// TIA Portal V16 export
// export: Created 2023-04-18T08:26:50.8983284Z, ExportSetting WithDefaults, DisplayName Totally Integrated Automation Portal, DisplayVersion V16, DisplayName TIA Portal Version Control Interface, DisplayVersion V16, DisplayName TIA Portal Openness, DisplayVersion V16, DisplayName SINAMICS Startdrive Advanced, DisplayVersion V16, DisplayName SINAMICS Startdrive G130, G150, S120, S150, SINAMICS MV, S210, DisplayVersion V16, DisplayName SINAMICS Startdrive G110M, G120, G120C, G120D, G120P, DisplayVersion V16, DisplayName STEP 7 Professional, DisplayVersion V16, DisplayName SIMATIC Energy Suite, DisplayVersion V16, DisplayName STEP 7 Safety, DisplayVersion V16, DisplayName WinCC Professional, DisplayVersion V16, DisplayName SIMATIC Visualization Architect, DisplayVersion V16
FUNCTION_BLOCK "IEQ"   // FB9, LAD
{ S7_Optimized_Access := 'TRUE' }
VERSION : 0.1
// stored: AutoNumber true, IsIECCheckEnabled false, IsRetainMemResEnabled false, MemoryReserve 100, SetENOAutomatically false, UDAEnableTagReadback false
   VAR_INPUT
      Fusible_R : Bool;
      Fusible_S : Bool;
      Fusible_T : Bool;
      "Fallo_ Tarjeta" : Bool;
      Seta : Bool;
      Fallo_Red : Bool;
      Ahorro_S0 : Bool;
      Ahorro_S1 : Bool;
      Directo_S0 : Bool;
      Directo_S1 : Bool;
      Nucleo_S0 : Bool;
      Nucleo_S1 : Bool;
      Tiristor : Int;
      Nucleo : Int;
   END_VAR
   VAR_OUTPUT
      alpha : Int;
      ventiladores : Bool;
      Ahorro_P0 : Bool;
      Ahorro_P1 : Bool;
      Directo_P0 : Bool;
      Directo_P1 : Bool;
      Nucleo_P0 : Bool;
      Nucleo_P1 : Bool;
   END_VAR
   VAR_IN_OUT
      AHM1 : "AHM1";
      IEQ : "IEQSY";
   END_VAR
   VAR
      Etapa_Emergencia : Int;
      Alpha_Conmutación : Bool;
   END_VAR
   VAR RETAIN
      Etapa : Int;
   END_VAR
   VAR
      S_Etapa : Int;
      Error : Int;
      Temporizadores : Struct
         T_E1 { S7_SetPoint := 'True'} : TON_TIME;
         T_E2 { S7_SetPoint := 'True'} : TON_TIME;
         T_E3 { S7_SetPoint := 'True'} : TON_TIME;
         T_E4 { S7_SetPoint := 'True'} : TON_TIME;
         T_E5 { S7_SetPoint := 'True'} : TON_TIME;
         T_E7 { S7_SetPoint := 'True'} : TON_TIME;
         T_SE1 { S7_SetPoint := 'True'} : TON_TIME;
         T_SE2 { S7_SetPoint := 'True'} : TON_TIME;
         T_SE3 { S7_SetPoint := 'True'} : TON_TIME;
         T_SE4 { S7_SetPoint := 'True'} : TON_TIME;
      END_STRUCT;
      F_TRIG_Seta { S7_SetPoint := 'True'} : F_TRIG;
      F_TRIG_Fusible_R { S7_SetPoint := 'True'} : F_TRIG;
      F_TRIG_Fusible_S { S7_SetPoint := 'True'} : F_TRIG;
      F_TRIG_Fusible_T { S7_SetPoint := 'True'} : F_TRIG;
      F_TRIG_Fallo_Red { S7_SetPoint := 'True'} : F_TRIG;
      R_TRIG_ETAPA { S7_SetPoint := 'True'} : R_TRIG;
      R_TRIG_BTN { S7_SetPoint := 'True'} : R_TRIG;
      F_TRIG_BTN { S7_SetPoint := 'True'} : F_TRIG;
      NormVal { ExternalAccessible := 'False'; ExternalVisible := 'False'; ExternalWritable := 'False'} : Real;
      message : String;
      showPopUp : Bool;
      ValHMI { ExternalAccessible := 'False'; ExternalVisible := 'False'; ExternalWritable := 'False'} : Int;
   END_VAR
BEGIN

REGION Network 1 (SCL)
   //*********************************************************************************************************************
   // Autor : Illya Kulinich
   // 
   // Descripción : 

   //*********************************************************************************************************************
END_REGION

REGION Network 2 (SCL): Flancos

   #F_TRIG_Seta(CLK :=#Seta);
   #F_TRIG_Fusible_R(CLK := #Fusible_R);
   #F_TRIG_Fusible_S(CLK := #Fusible_S);
   #F_TRIG_Fusible_T(CLK := #Fusible_T);
   #F_TRIG_Fallo_Red(CLK := #Fallo_Red);
   #R_TRIG_BTN(CLK:=#IEQ.Conmutación.BTN);
   #F_TRIG_BTN(CLK := #IEQ.Conmutación.BTN);
END_REGION

REGION Network 3 (SCL): Conversión de temperatura en real

   #IEQ.Temperatura.Tiristores := (INT_TO_REAL(#Tiristor)) * 0.1;
   #IEQ.Temperatura.Nucleo  := (INT_TO_REAL(#Nucleo)) * 0.1;
END_REGION

REGION Network 4 (SCL): Declaración de temporizadores

       //
       #Temporizadores.T_SE1(IN := #Etapa_Emergencia = 1,
                             PT := T#1S);
       #Temporizadores.T_SE2(IN := #Etapa_Emergencia = 2,
                             PT := T#1S);
       #Temporizadores.T_SE3(IN := #Etapa_Emergencia = 3,
                             PT := T#1S);
       #Temporizadores.T_SE4(IN := #Etapa_Emergencia = 4,
                             PT := T#1S);

       //******************************************************************     
       #Temporizadores.T_E1(IN := #Etapa = 1,
                             PT := T#2.5s);
       #Temporizadores.T_E2(IN := #Etapa = 2,
                             PT := T#2.5s);
       #Temporizadores.T_E3(IN := #Etapa = 3,
                             PT := T#2.5s);
       #Temporizadores.T_E4(IN := #Etapa = 4,
                             PT := T#2.5s);
       #Temporizadores.T_E5(IN := #Etapa = 5,
                             PT := T#2.5s);
       #Temporizadores.T_E7(IN := #Etapa = 7,
                             PT := T#2.5s);
END_REGION

REGION Network 5 (SCL): Estado de Conmutación
   // Ahorro
   IF #Ahorro_S0 = 0 AND #Ahorro_S1 = 1 AND
       #Directo_S0 = 1 AND #Directo_S1 = 0 AND
       #Nucleo_S0 = 0 AND #Nucleo_S1 = 1 THEN
       #IEQ.Conmutación.Status := 'Ahorro';
   END_IF;


   // transición
   IF #Ahorro_S0 = 0 AND #Ahorro_S1 = 1 AND
       #Directo_S0 = 0 AND #Directo_S1 = 1 AND
       #Nucleo_S0 = 0 AND #Nucleo_S1 = 1 THEN
       #IEQ.Conmutación.Status  := 'Conmutando...';
   END_IF;

   // Directo 
   IF #Ahorro_S0 = 1 AND #Ahorro_S1 = 0 AND
       #Directo_S0 = 0 AND #Directo_S1 = 1 AND
       #Nucleo_S0 = 1 AND #Nucleo_S1 = 0 THEN
       #IEQ.Conmutación.Status  := 'Directo';

   END_IF;
END_REGION

REGION Network 6 (SCL): Seguridad

   IF (#F_TRIG_Fusible_R.Q OR #F_TRIG_Fusible_S.Q OR #F_TRIG_Fusible_T.Q) AND  #IEQ.Conmutación.BTN = 1  THEN
       #Etapa_Emergencia := 99;

   END_IF;

   IF #F_TRIG_Seta.Q AND #IEQ.Conmutación.BTN= 1 THEN
       #Etapa_Emergencia := 99;
   END_IF;

   IF  #IEQ.Temperatura.Tiristores >= 75.0 OR  #IEQ.Temperatura.Nucleo >= 120.0 AND #IEQ.Conmutación.BTN = 1 THEN
       #Etapa_Emergencia := 99;

   END_IF;

   IF #F_TRIG_Fallo_Red.Q AND #IEQ.Conmutación.BTN= 1 THEN
       #Etapa_Emergencia := 99;
   END_IF;



   // IF NOT #Fusible_R OR NOT #Fusible_S OR NOT #Fusible_T OR
   //     NOT #Seta OR
   //     NOT #Fallo_Red OR
   //     NOT (#IEQ.Temperatura.Tiristores < 50.0 AND #IEQ.Temperatura.Nucleo < 60.0) THEN
   IF #Fallo_Red THEN
       #Error := 1;
       #message := 'Error en la red';
       // pop up fallo fusibles
       // DTL timestamp
   ELSE
       #Error := 0;
   END_IF;

   IF #Error = 1 THEN
       #IEQ.Conmutación.BTN := 0;
       #IEQ.Alpha.Input_Value := 100;
       #showPopUp := 1;
   ELSE
       #Error := 0;
   END_IF;


   (* IF NOT  #Fallo_Red  THEN
       #IEQ.Conmutación.BTN := 0;
       // pop up fallo de red 
       // DTL timestamp
   END_IF;

   (* IF #"Fallo_ Tarjeta" THEN
       #IEQ.Conmutación.BTN := 0;
       // pop up tarjeta de tiristores
       // DTL timestamp
   END_IF; *)

   IF NOT (  < 50.0  OR  #IEQ.Temperatura.Tiristores < 50.0  OR  < 50.0  AND #IEQ.Temperatura.Nucleo < 60.0) AND #IEQ.Conmutación.BTN =1 THEN
       #IEQ.Conmutación.BTN := 0;
       // pop up temperatura 
       // DTL timestamp
   END_IF;
   *)
END_REGION

REGION Network 7 (SCL): Secuencia de emergencia





       IF #Etapa_Emergencia = 99 THEN

           #Etapa := 0;
           #Etapa_Emergencia := 1;

           #IEQ.Conmutación.BTN := 0;
           #Alpha_Conmutación := 1;

           #Ahorro_P0 := 0;
           #Ahorro_P1 := 1;
           #Directo_P0 := 0;
           #Directo_P1 := 1;
           #Nucleo_P0 := 0;
           #Nucleo_P1 := 1;
       END_IF;

       IF #Etapa_Emergencia = 1 AND #Temporizadores.T_SE1.Q THEN
           #Etapa_Emergencia := 2;
           #Alpha_Conmutación := 1;
           #Ahorro_P0 := 1;
           #Ahorro_P1 := 0;
           #Directo_P0 := 0;
           #Directo_P1 := 1;
           #Nucleo_P0 := 0;
           #Nucleo_P1 := 1;
       END_IF;

       IF #Etapa_Emergencia = 2 AND #Temporizadores.T_SE2.Q THEN
           #Etapa_Emergencia := 3;
           #Alpha_Conmutación := 1;
           #Ahorro_P0 := 1;
           #Ahorro_P1 := 0;
           #Directo_P0 := 0;
           #Directo_P1 := 1;
           #Nucleo_P0 := 1;
           #Nucleo_P1 := 0;

       END_IF;

       IF #Etapa_Emergencia = 3 AND #Temporizadores.T_SE3.Q THEN
           #Etapa_Emergencia := 0;
           #Etapa := 3;
       END_IF;
END_REGION

REGION Network 8 (SCL): Conmutación


       IF #Etapa = 99 THEN
           #Etapa := 1;

           #Alpha_Conmutación := 1;
           #Ahorro_P0 := 0;
           #Ahorro_P1 := 1;
           #Directo_P0 := 0;
           #Directo_P1 := 1;
           #Nucleo_P0 := 0;
           #Nucleo_P1 := 1;

       END_IF;

       IF #Etapa = 1 AND #Temporizadores.T_E1.Q THEN
           #Etapa := 2;
           #Alpha_Conmutación := 1;
           #Ahorro_P0 := 1;
           #Ahorro_P1 := 0;
           #Directo_P0 := 0;
           #Directo_P1 := 1;
           #Nucleo_P0 := 0;
           #Nucleo_P1 := 1;
       END_IF;

       IF #Etapa = 2 AND #Temporizadores.T_E2.Q THEN // Directo
           #Etapa := 3;
           #Alpha_Conmutación := 1;
           #Ahorro_P0 := 1;
           #Ahorro_P1 := 0;
           #Directo_P0 := 0;
           #Directo_P1 := 1;
           #Nucleo_P0 := 1;
           #Nucleo_P1 := 0;


       END_IF;


       IF #Etapa = 3 AND #Temporizadores.T_E3.Q AND #R_TRIG_BTN.Q AND #Error = 0 THEN
           #Etapa := 4;
           #Alpha_Conmutación := 1;
           #Ahorro_P0 := 1;
           #Ahorro_P1 := 0;
           #Directo_P0 := 0;
           #Directo_P1 := 1;
           #Nucleo_P0 := 0;
           #Nucleo_P1 := 1;

       END_IF;

       IF #Etapa = 4 AND #Temporizadores.T_E4.Q THEN
           #Etapa := 5;
           #Alpha_Conmutación := 1;
           #Directo_P0 := 0;
           #Directo_P1 := 1;

           #Ahorro_P0 := 0;
           #Ahorro_P1 := 1;

           #Nucleo_P0 := 0;
           #Nucleo_P1 := 1;

       END_IF;

       IF #Etapa = 5 AND #Temporizadores.T_E5.Q THEN
           #Etapa := 6;
           #Alpha_Conmutación := 0;
           #Ahorro_P0 := 0;
           #Ahorro_P1 := 1;
           #Directo_P0 := 1;
           #Directo_P1 := 0;
           #Nucleo_P0 := 0;
           #Nucleo_P1 := 1;

       END_IF;

       IF #Etapa = 6 AND #F_TRIG_BTN.Q THEN
           #Etapa := 99;
           #Alpha_Conmutación := 1;
       END_IF;
END_REGION

REGION Network 9 (SCL)

   REGION Definición de las condiciones de protección frente a valores no desados

       // si alguna de estas condiciónes son verdaderas el alpha setpoint pasa a 100
       IF #Alpha_Conmutación = 0 AND
           (#AHM1."Parametros Basicos"."40007 - Tension y Energia".PF1 < #IEQ.Alpha.RestriccionesAlpha.PF_Min_Alpha OR
           #AHM1."Parametros Basicos"."40007 - Tension y Energia".PF2 < #IEQ.Alpha.RestriccionesAlpha.PF_Min_Alpha OR
           #AHM1."Parametros Basicos"."40007 - Tension y Energia".PF3 < #IEQ.Alpha.RestriccionesAlpha.PF_Min_Alpha OR

           #AHM1."Harmonic data"."40529 - Distorsion Armonica V y A"."THD-V1" > #IEQ.Alpha.RestriccionesAlpha.Thd_V_Max OR
           #AHM1."Harmonic data"."40529 - Distorsion Armonica V y A"."THD-V2" > #IEQ.Alpha.RestriccionesAlpha.Thd_V_Max OR
           #AHM1."Harmonic data"."40529 - Distorsion Armonica V y A"."THD-V3" > #IEQ.Alpha.RestriccionesAlpha.Thd_V_Max OR

           #AHM1."Harmonic data"."40529 - Distorsion Armonica V y A"."THD-I1" > #IEQ.Alpha.RestriccionesAlpha.Thd_A_Max OR
           #AHM1."Harmonic data"."40529 - Distorsion Armonica V y A"."THD-I2" > #IEQ.Alpha.RestriccionesAlpha.Thd_A_Max OR
           #AHM1."Harmonic data"."40529 - Distorsion Armonica V y A"."THD-I3" > #IEQ.Alpha.RestriccionesAlpha.Thd_A_Max)
       THEN
           ;
           // si el pf y el thd en voltaje y corriente baja de x   alpha entra en error pon el valor a 100 ->  alpha a 100% = 5 V = 13834

           #IEQ.Alpha.AlphaEntero := 27648;
           #IEQ.Alpha.Status := 'Condiciones de red no se cumplen alpha es 100';


       END_IF;

   END_REGION

   REGION Definicion del correcto funcionamiento de alpha


       /// Si todas las condiciones son correctas  escalamos el valor del ewon o de la pantalla hmi 

       IF #Alpha_Conmutación = 0 AND
           (*NOT*)(#AHM1."Parametros Basicos"."40007 - Tension y Energia".PF >= #IEQ.Alpha.RestriccionesAlpha.PF_Min_Alpha OR

           #AHM1."Harmonic data"."40529 - Distorsion Armonica V y A"."THD-V1" <= #IEQ.Alpha.RestriccionesAlpha.Thd_V_Min OR
           #AHM1."Harmonic data"."40529 - Distorsion Armonica V y A"."THD-V2" <= #IEQ.Alpha.RestriccionesAlpha.Thd_V_Min OR
           #AHM1."Harmonic data"."40529 - Distorsion Armonica V y A"."THD-V3" <= #IEQ.Alpha.RestriccionesAlpha.Thd_V_Min OR

           #AHM1."Harmonic data"."40529 - Distorsion Armonica V y A"."THD-I1" <= #IEQ.Alpha.RestriccionesAlpha.Thd_A_Min OR
           #AHM1."Harmonic data"."40529 - Distorsion Armonica V y A"."THD-I2" <= #IEQ.Alpha.RestriccionesAlpha.Thd_A_Min OR
           #AHM1."Harmonic data"."40529 - Distorsion Armonica V y A"."THD-I3" <= #IEQ.Alpha.RestriccionesAlpha.Thd_A_Min)
       THEN

           // alpha esta en OK pon el valor de la variable al que venga del Ewon (95%)  
           IF #IEQ.Alpha.Input_Value >= 85 AND #IEQ.Alpha.Input_Value <= 100 THEN
               #ValHMI := #IEQ.Alpha.Input_Value;
           ELSE
               #ValHMI := #IEQ.Alpha.Input_Value := 100;

           END_IF;

           #NormVal := NORM_X(MIN := 0, VALUE := #ValHMI, MAX := 100);
           #IEQ.Alpha.AlphaEntero := SCALE_X(MIN := 0, VALUE := #NormVal, MAX := 27648); // son 4.95V -> 13824 intento de ajustar el valor al de la tarjeta
           #IEQ.Alpha.Status := 'Condiciones de red no se cumplen alpha es 100';
       END_IF;

   END_REGION


   REGION

       IF #Alpha_Conmutación = 1 THEN 
           #IEQ.Alpha.AlphaEntero := 27648;
           #IEQ.Alpha.Status := 'Conmutando/Directo';
       END_IF;

   END_REGION


   #alpha := #IEQ.Alpha.AlphaEntero;
END_REGION

REGION Network 10 (SCL)
   IF #IEQ.Ventilación.testeo = 1 THEN
       #ventiladores := 1;

   END_IF;


   IF NOT #IEQ.Ventilación.testeo AND ( #IEQ.Temperatura.Tiristores > 35  OR #IEQ.Temperatura.Nucleo > 80) THEN
       #ventiladores := 1;

   END_IF;


   IF NOT #IEQ.Ventilación.testeo AND ( #IEQ.Temperatura.Tiristores < 30 AND #IEQ.Temperatura.Nucleo < 70) THEN
       #ventiladores := 0;

   END_IF;
END_REGION
END_FUNCTION_BLOCK
